// TIA Portal V19 export
TYPE "lexchangetray_typeUnEmn_toConstraintWorkstationReq"
// Type: Bool
// stored: Access Published
   STRUCT
      transferEnable : Bool;   // Manual mode parameters for axis control interface
      unConstraint : Bool;   // Manual mode parameters for axis control interface
      Constraint : Bool;   // Manual mode parameters for axis control interface
   END_STRUCT;
END_TYPE
